PROGRAM ResetAxes
VAR
	resetstate				:INT	:= 0;
END_VAR

CASE resetstate OF
	0:
	IF GVL_MOTION.EXT_CTR.AxesReset THEN
		GVL_MOTION.EXT_CTR.AxesReset		:= FALSE;
		GVL_MOTION.HomingState				:= 0;
		GVL_MOTION.xCon.Execute_MREL		:= FALSE;
		//GVL_MOTION.HardStopState			:= 0;
		GVL_MOTION.xCon.Execute_HOME		:= FALSE;
		GVL_MOTION.xcCon.Execute_HOME		:= FALSE;
		GVL_MOTION.xCon.Execute_HALT		:= FALSE;
		GVL_MOTION.xcCon.Execute_HALT		:= FALSE;
		GVL_MOTION.xCon.Execute_RES 		:= TRUE;
		IF NOT GVL_MOTION.xOut.AxisCoupled THEN
			GVL_MOTION.xcCon.Execute_RES	:= TRUE;
		END_IF
		GVL_MOTION.yCon.Execute_HOME		:= FALSE;
		GVL_MOTION.yCon.Execute_HALT		:= FALSE;
		GVL_MOTION.yCon.Execute_RES 		:= TRUE;
		GVL_MOTION.zCon.Execute_HOME		:= FALSE;
		GVL_MOTION.zCon.Execute_HALT		:= FALSE;
		GVL_MOTION.zCon.Execute_RES 		:= TRUE;
		resetstate							:= 1;
	END_IF	
	1:
		GVL_MOTION.xCon.Execute_RES 		:= FALSE;
		GVL_MOTION.xcCon.Execute_RES		:= FALSE;
		GVL_MOTION.yCon.Execute_RES 		:= FALSE;
		GVL_MOTION.zCon.Execute_RES 		:= FALSE;
		resetstate							:= 0;
END_CASE

END_PROGRAM

(* stored: Version 1.1.0.1, ProductVersion 3.1.4026.18
   POU ResetAxes: Id {c54c8a7f-9baf-498e-9f01-ec7612f9cf7e}, SpecialFunc None *)
